{attribute addProperty BoxType "EL2262-0000-0002"}
{attribute addProperty Id "Cycle_Counter0AT %Q*UINT162"}
{attribute addProperty CRC "812659932"}
{attribute addProperty SizeInBites "16"}
{attribute addProperty SizeInBytes "2"}
TYPE CycCount0_307034DC :
STRUCT
	{attribute addProperty Name "Cycle_Counter0"}
	Cycle_Counter0 AT %Q* : UINT;
END_STRUCT
END_TYPE

(* stored: Version 1.2.0.0, ProductVersion 3.1.4024.9
   DUT CycCount0_307034DC: Id {2b041f17-710e-4319-92ac-dfe4345514d4} *)
